# EPICS substitutions: elioApp/Db/EL4008.substitutions
file EL4008.template { pattern
{ CHAN	}
{ 1	}
{ 2	}
{ 3	}
{ 4	}
{ 5	}
{ 6	}
{ 7	}
{ 8	}
}
